FUNCTION_BLOCK FB_TMCM1140_Power
VAR_INPUT
	bExecute : BOOL;
END_VAR
VAR_OUTPUT
	bBusy 		: BOOL;
	bError 		: BOOL;
	nErrorId 	: ERRORID;	
END_VAR
VAR_IN_OUT
	pHwRef : POINTER TO FB_HwRefTMCM1140;
END_VAR
VAR
	nState 		: USINT;
	nStateNext 	: USINT;
	fbSdoWrite	: FB_SDO_WRITE;
	nDataDigiOut: DINT;
END_VAR

IF bExecute THEN
	IF nState = 0 THEN
		bBusy := TRUE; 
		CASE pHwRef^.M_GetDS402State() OF
			E_CoDS402States.DS402STATE_Fault:
				pHwRef^.nControlword := 153;	//Reset error
				nState := 1;
			E_CoDS402States.DS402STATE_SwitchOnDisabled:
				nState := 1;
			E_CoDS402States.DS402STATE_ReadyToSwitchOn:
				pHwRef^.nControlword := 0;	//Transition 7 in DS402 statemachine -> geht in Switch on disabled
				nState := 1;
			E_CoDS402States.DS402STATE_SwitchedOn:
				pHwRef^.nControlword := 0;	//Transition 10 in DS402 statemachine -> geht in Switch on disabled
				nState := 1;
			E_CoDS402States.DS402STATE_OperationEnabled:
				pHwRef^.nControlword := 0;	//Shutdown
				nState := 1;
			E_CoDS402States.DS402STATE_NotReadyToSwitchOn:	//Statusword wahrscheinlich nicht gemappt
				nErrorId := E_ErrorIdDS402.ERRORID_NotReadyToSwitchOn;
				nState := 99;
		END_CASE
	END_IF
	
	CASE nState OF
		1:	//Hier sollte noch ein Timeout eingebaut werden?
			IF pHwRef^.M_GetDS402State() = E_CoDS402States.DS402STATE_SwitchOnDisabled THEN
				//max. current
				fbSdoWrite.nIndex := 16#2003;
				fbSdoWrite.nSubIndex := 0;
				fbSdoWrite.nDataLength := 1;
				fbSdoWrite.nData := pHwRef^.P_nMaxCurrentConverted;
				nState := 40;
				nStateNext := 2;
			END_IF
			
		2:	//Hold current
			fbSdoWrite.nIndex := 16#2004;
			fbSdoWrite.nSubIndex := 0;
			fbSdoWrite.nDataLength := 1;
			fbSdoWrite.nData := pHwRef^.P_nHoldCurrentConverted;
			nState := 40;
			nStateNext := 3;

		3:	//Switch parameters (Endlagen)		
			fbSdoWrite.nIndex := 16#2005;
			fbSdoWrite.nSubIndex := 0;
			fbSdoWrite.nDataLength := 4;
			fbSdoWrite.nData := pHwRef^.P_nSwitchConfig;
			nState := 40;
			nStateNext := 4;		
			
		4:	//Brake deaktivieren
			fbSdoWrite.nIndex := 16#200C;
			fbSdoWrite.nSubIndex := 2;
			fbSdoWrite.nDataLength := 1;
			fbSdoWrite.nData := 0;
			nState := 40;
			nStateNext := 5;

		5:	//Position Windows setzen
			fbSdoWrite.nIndex := 16#6067;
			fbSdoWrite.nSubIndex := 0;
			fbSdoWrite.nDataLength := 4;
			fbSdoWrite.nData := 100;
			nState := 40;
			nStateNext := 6;
			
		6:	//Velocity Dimension Index -> Intern (damit die folgenden Werte geschrieben werden können)
			fbSdoWrite.nIndex := 16#208C;
			fbSdoWrite.nSubIndex := 0;
			fbSdoWrite.nDataLength := 1;
			fbSdoWrite.nData := E_TMCM_VeloDim.INTERN;
			nState := 40;
			nStateNext := 7;
			
		7:	//Microstep Resolution
			fbSdoWrite.nIndex := 16#2000;
			fbSdoWrite.nSubIndex := 0;
			fbSdoWrite.nDataLength := 1;
			fbSdoWrite.nData := pHwRef^.P_nMicrostepResolConverted;
			nState := 40;
			nStateNext := 31;
			
		31:	//FullStep Resolution
			fbSdoWrite.nIndex := 16#2001;
			fbSdoWrite.nSubIndex := 0;
			fbSdoWrite.nDataLength := 2;
			fbSdoWrite.nData := pHwRef^.P_nFullStepRevo;
			nState := 40;
			nStateNext := 8;
			
		8:	//Pulse Divisor
			fbSdoWrite.nIndex := 16#2086;
			fbSdoWrite.nSubIndex := 0;
			fbSdoWrite.nDataLength := 1;
			fbSdoWrite.nData := pHwRef^.P_nPulseDivisor;
			nState := 40;
			nStateNext := 9;
			
		9:	//Ramp Divisor
			fbSdoWrite.nIndex := 16#2085;
			fbSdoWrite.nSubIndex := 0;
			fbSdoWrite.nDataLength := 1;
			fbSdoWrite.nData := pHwRef^.P_nRampDivisor;
			nState := 40;
			nStateNext := 10;
			
		10:	//Digital out mask
			fbSdoWrite.nIndex := 16#2703;
			fbSdoWrite.nSubIndex := 2;
			fbSdoWrite.nDataLength := 4;
			nDataDigiOut.16 := pHwRef^.P_bSetDigiOut0;
			nDataDigiOut.17 := pHwRef^.P_bSetDigiOut1;
			fbSdoWrite.nData := nDataDigiOut;
			nState := 40;
			nStateNext := 11;

		11:	//Set digital out
			fbSdoWrite.nIndex := 16#2703;
			fbSdoWrite.nSubIndex := 1;
			fbSdoWrite.nDataLength := 4;
			fbSdoWrite.nData := nDataDigiOut;
			nState := 40;
			nStateNext := 12;
			
		12:	//Change to "Ready to Switched on"
			pHwRef^.nControlword := 6;
			nState := 13;
			
		13:	IF pHwRef^.M_GetDS402State() = E_CoDS402States.DS402STATE_ReadyToSwitchOn THEN
				pHwRef^.nControlword := 7;	//Change to "Switched on"
				nState := 14;
			ELSIF pHwRef^.M_GetDS402State() = E_CoDS402States.DS402STATE_Fault THEN
				nErrorId := E_ErrorIdDS402.ERRORID_FaultState;
				nState := 99;
			END_IF
			
		14:	IF pHwRef^.M_GetDS402State() = E_CoDS402States.DS402STATE_SwitchedOn THEN
				pHwRef^.nControlword := 15;	//Change to "Operation enable"
				nState := 15;
			ELSIF pHwRef^.M_GetDS402State() = E_CoDS402States.DS402STATE_Fault THEN
				nErrorId := E_ErrorIdDS402.ERRORID_FaultState;
				nErrorId := 232;
				nState := 99;
			END_IF
			
		15:	IF pHwRef^.M_GetDS402State() = E_CoDS402States.DS402STATE_OperationEnabled THEN
				nState := 80;
			ELSIF pHwRef^.M_GetDS402State() = E_CoDS402States.DS402STATE_Fault THEN
				nErrorId := E_ErrorIdDS402.ERRORID_FaultState;
				nErrorId := 232;
				nState := 99;
			END_IF
	END_CASE
	
	//Sdo senden
	IF nState = 40 THEN
		fbSdoWrite(sADSNetID:= pHwRef^.P_sAdsNetId, nPortNr:= pHwRef^.P_nAdsPort, bExecute:= TRUE);
		IF NOT fbSdoWrite.bBusy THEN
			IF fbSdoWrite.bError THEN
				nErrorId := fbSdoWrite.nAdsErrorId;
				nState := 99;
			ELSE
				nState := nStateNext;
			END_IF
			fbSdoWrite(bExecute:= FALSE);
		END_IF		
	END_IF
	
	IF nState >= 80 THEN
		bBusy := FALSE;
		IF nState = 99 THEN
			bError := TRUE;
		END_IF
	END_IF

ELSE
	bBusy := FALSE;
	bError := FALSE;
	nErrorId := 0;
	nState := 0;	
END_IF

END_FUNCTION_BLOCK

(* stored: Version 1.1.0.1, ProductVersion 3.1.4024.14
   POU FB_TMCM1140_Power: Id {74546f5f-43e7-4a2d-ac41-18d8406b798a}, SpecialFunc None *)
